FUNCTION_BLOCK EventLoggerManager IMPLEMENTS EventManager
VAR
	eventLogger : FB_TcEventLogger;
END_VAR

METHOD ClearAll
VAR_INPUT
END_VAR
eventLogger.ClearAlarms(0, TRUE, 0);
END_METHOD

END_FUNCTION_BLOCK

(* stored: Version 1.1.0.1
   POU EventLoggerManager: Id {92790c3e-d2fe-06db-267a-42aa72ce045d}, SpecialFunc None
   Method ClearAll: Id {28e95231-a3ef-0a9a-1795-305279e64ada} *)
